{attribute 'linkalways'} 
{attribute 'no_explicit_call' := 'This FB is a CLASS and must be accessed using methods or properties'}
{attribute 'enable_dynamic_creation'}
FUNCTION_BLOCK Node_F_VN_GetAt_TcVnVector2_INT EXTENDS VisionNode
VAR
    ipContainer : _ITcVnContainer;
    aElement : _TcVnVector2_INT;
    nIndex : _ULINT(0);
    hrPrev : _HRESULT(S_OK);
    hresult : _HRESULT(S_OK);
END_VAR

METHOD PUBLIC  Clone : I_Node
VAR
	pNode : POINTER TO Node_F_VN_GetAt_TcVnVector2_INT;
END_VAR
pNode := __NEW(Node_F_VN_GetAt_TcVnVector2_INT);
Clone := pNode^;
END_METHOD

METHOD FB_init : BOOL
VAR_INPUT
	bInitRetains : BOOL; // if TRUE, the retain variables are initialized (warm start / cold start)
	bInCopyCode : BOOL;  // if TRUE, the instance afterwards gets moved into the copy code (online change)
END_VAR
AddInput('ipContainer', ipContainer);
AddInput('nIndex', nIndex);
AddInput('hrPrev', hrPrev);
AddOutput('aElement', aElement);
AddOutput('hresult',hresult);
END_METHOD

METHOD PROTECTED OnExecute : HRESULT
hresult.Value := F_VN_GetAt_TcVnVector2_INT(
    ipContainer := ipContainer.Value,
    aElement := aElement.Value,
    nIndex := nIndex.Value,
    hrPrev:= hrPrev.Value);
END_METHOD

METHOD PUBLIC PreExecutionCheck
VAR_INPUT
	Check : I_PreExecutionChecks;
END_VAR
Check.IsTrue(ipContainer.IsValid, 'ipContainer must be a valid container');
Check.IsTrue(ipContainer.HasType(TC_GLOBAL_CONST_LIST.ContainerType_Vector_TcVnVector2_INT), 'ipContainer contains incorrect type');
END_METHOD

END_FUNCTION_BLOCK

(* stored: Version 1.1.0.1, ProductVersion 3.1.4024.13
   POU Node_F_VN_GetAt_TcVnVector2_INT: Id {b9263e00-0f6e-4bfa-922f-1131a923d35b}, SpecialFunc None
   Folder Constructor: Id {8a05a779-45c1-4012-997e-6a544be0a34e}
   Method Clone: Id {709cdbf7-d338-483e-8563-5f5510c560ca}
   Method FB_init: Id {0bd3de4b-1549-4624-aff3-5b6414a14eb8}
   Method OnExecute: Id {6f11e0d3-c4d2-4c02-9ea2-8024092e2836}
   Method PreExecutionCheck: Id {ab1df4d4-abc1-4f40-98f4-56fdf256bb4f} *)
